// TIA Portal V18 export
ORGANIZATION_BLOCK "Time error interrupt"   // OB80, LAD, TimeErrorInterrupt
{ S7_Optimized_Access := 'TRUE' }
VERSION : 0.1
// stored: IsIECCheckEnabled false, SetENOAutomatically false
   VAR_INPUT
      Fault_ID : Byte;   // Fault identifier
      Csg_OBnr : OB_ANY;   // Number of OB causing the error
      Csg_Prio : UInt;   // Priority of OB causing the error
   END_VAR
BEGIN
END_ORGANIZATION_BLOCK
